Staubli VAL3: start.pgx

program start()
begin
  // Initialisation
  call init()

  // tPosition : envoi position toutes les 40ms (sync)
  taskCreateSync sTaskPos, 0.040, bOvrPosition, tPosition()
  wait(taskStatus(sTaskPos) == 1)

  // tCommande : reception des commandes
  taskCreate sTaskCmd, 100, tCommande()
  wait(taskStatus(sTaskCmd) == 1)

  // tRobot : execution des mouvements
  taskCreate sTaskRobot, 100, tRobot()
  wait(taskStatus(sTaskRobot) == 1)

  // Surveillance des overruns
  while true
    if nPrevOvrPos != nOvrPos
      logMsg("Overrun dans la tache " + sTaskPos)
      nPrevOvrPos = nOvrPos
    endIf
    delay(0)
  endWhile
end
